(* PLC project Generated.project, CODESYS CODESYS V3.5 SP19 Patch 1 *)
(* stored: creationDateTime 2026-11-16T05:01:26.673404, modificationDateTime 2026-11-16T05:01:26.673404 *)

(* DOC: DOC/AF/AF_Partie-13_Fonction_Simulation_v2.5.md Modele dynamique M3 confine au SimBench. *)
FUNCTION_BLOCK FB_Sim_Translation
  VAR_INPUT
    Enable : BOOL;
    ReqTremie : BOOL;
    ReqMaintenance : BOOL;
    SpeedTgt_Pct : REAL;
    PosTremie_M : REAL := 0;  (* T301/L1 — SOURCE UNIQUE : le banc ne porte AUCUNE position ni echelle propre. Positions capteurs = reglages machine (GVL_PERSISTENT._TranslationPos*_M) et gain = gain EFFECTIVEMENT consomme par l'estimateur (PRG_05 FB_Translation_OdometryGain.GainActive), passes par PRG_02 -> FB_SimBench. Vitesse chariot = sens x gain x frequence. Historique : l'ancienne echelle en dur (30 m / FullTravelTimeS / 40 Hz) a diverge du gain reel (T360/T361, sauts de 4 a 9 m) — doublon supprime, gate G518 anti-retour. --> [CFG] Position capteur Tremie (m) *)
    PosPV_M : REAL := 1.5;  (* --> [CFG] Position capteur PV (m) *)
    PosP2_M : REAL := 3.5;  (* --> [CFG] Position capteur P2 (m) *)
    PosP1_M : REAL := 5;  (* --> [CFG] Position capteur P1 (m) *)
    PosMaintenance_M : REAL := 10;  (* --> [CFG] Position capteur Maintenance (m) *)
    GainMetersPerHzSec : REAL := 0.02;  (* --> [CFG] Gain odometrique effectif, m/(Hz.s) *)
    EndStopMargin_M : REAL := 0.5;  (* Distance capteur extreme -> butee mecanique (seule donnee propre au banc : physique du rail). Bornee a CST_MinEndStopMargin_M pour que le capteur extreme reste franchissable. *)
    BrakeReleaseCmd : BOOL := TRUE;
    MaxFreq_Hz : REAL := 50;  (* ECHELLE DE LA CONSIGNE. PRG_02 envoie SpeedCmd_Pct = f / 50 Hz x 100 : le simulateur reconvertit avec le MEME maximum, sinon 20 Hz reels (40 %) deviendraient 16 Hz simules. Maximum = GVL_PERSISTENT._TranslationMaxFreq_Hz (50 Hz), passe par FB_SimBench (CST_M3MaxFreq_Hz, egalite verifiee par G518). Ne pas confondre avec l'ancienne echelle (40 Hz) : echelle ODOMETRIQUE (gain 0,02 m/(Hz.s)). *)
    SpeedFactor : REAL := 1;  (* ACCELERATION DU BANC (confort d'essai). Le chariot avance SpeedFactor fois plus vite ET la frequence RETOURNEE au PLC est multipliee d'autant : l'estimateur (f x gain) suit exactement le chariot, sans saut de recalage, et le ratio publie reste 0,02 m/(Hz.s) (G518). Borne 1..5. 1,0 = dynamique reelle. Le frein et la memoire de sens restent sur la frequence physique du variateur simule. *)
    AccelRate_HzPerS : REAL := 20;
    DecelRate_HzPerS : REAL := 25;  (* pente d'arret relevee sur trace reelle (rampe variateur / rampe PLC) *)
    DriveTimeConstantS : REAL := 0.15;
    BrakeOpenDelayS : REAL := 0.1;
    BrakeCloseDelayS : REAL := 0.09;
    BrakeContactDelayS : REAL := 0.01;
    BrakeFaultCloseWhileRunning : BOOL := FALSE;  (* FAUTE EXPLICITE frein M3 — defaut FALSE : reproduit le defaut terrain « frein ferme alors que le variateur retourne encore 10,00 Hz » (trace 2026-09-04, 26,437 s, State.ErrorId=64). La garde nominale 0,5 Hz du frein n'est pas modifiee. *)
    BrakeFaultCloseDelay_S : REAL := 0;
    BrakePhysicalActive : BOOL := FALSE;  (* L3 — FREIN PHYSIQUE (2026-10-28). FALSE = historique (frein ne retombe que sous 0,5 Hz, arret instantane). TRUE = frein a manque de courant reel : retombe CloseDelay apres la coupure bobine QUELLE QUE SOIT la vitesse, puis le chariot decelere sur le frein (BrakeDecel_Mps2) ; frein serre = chariot bloque meme si le variateur pousse. defaut FB = historique ; GVL_Simulation.SimM3BrakePhysicalActive = TRUE (source unique) *)
    BrakeDecel_Mps2 : REAL := 2;  (* HYPOTHESE : 0,4 m/s (20 Hz) -> arret ~0,2 s / ~4 cm *)
    CartFreeActive : BOOL := FALSE;  (* L4 — CHARIOT LIBRE (2026-10-28). FALSE = historique (chariot esclave de la frequence). TRUE = quand le frein est OUVERT et que le variateur n'applique plus de couple (mot a 0 et rampe variateur terminee), le chariot n'est plus tenu : il garde sa vitesse et subit la poussee de la benne suspendue (rapport de masse x g x angle), la pente et le frottement de roulement. Valeurs = HYPOTHESES, sans mesure terrain. *)
    LoadMassRatio : REAL := 0.5;  (* masse benne / masse totale chariot+benne *)
    RollingFriction_Mps2 : REAL := 0.3;  (* FEM 1.001 : frottement global galets + reducteur accouple *)
    StaticFriction_Mps2 : REAL := 0.35;  (* Seuil de decollement statique (anti-pompage pendulaire) *)
    Slope_Mps2 : REAL := 0;  (* composante de pente, + vers Maintenance *)
    SensorCamDropoutActive : BOOL := FALSE;  (* L5 — came capteurs (vu -> perdu -> retrouve -> fixe), appliquee aux 5 capteurs. *)
    SensorCamDropoutStart_M : REAL := 0.02;
    SensorCamDropoutWidth_M : REAL := 0.04;
    SuspendedLoadLength_M : REAL := 1.5;
    SuspendedLoadDamping : REAL := 0.35;
    LoadReactionGain_Mps2 : REAL := 0.2;
    EndStopRecoilMax_M : REAL := 0;  (* BUTEE MECANIQUE — recul borne apres arret serre. 0.0 (defaut) conserve EXACTEMENT le comportement historique : position ET vitesse figees a la butee (decision de review tracee, correctif « contact rigide »). > 0 : l'inertie du chariot reste absorbee par la butee, MAIS la reaction de la charge peut ressortir le chariot de la zone capteur — comportement observe sur la trace terrain du 2026-09-04 a 26,437 s (Tremie actif 1 echantillon puis perdu definitivement). Valeur SYNTHETIQUE, en attente de mesure terrain. *)
    LoadFrequencyDroopGain_Hz : REAL := 0.5;
    SensorJitterAmplitude_M : REAL := 0.01;
    SensorStabilizationS : REAL := 1;
    SensorElectricalDelayS : REAL := 0.01;
    SensorIntermittenceActive : BOOL := FALSE;
    SensorLoadAngleTriggerRad : REAL := 0.01;
    SensorScenarioSeed : UDINT := 3001;
    SensorHysteresis_M : REAL := 0.02;
    SensorIntermittencePeriodS : REAL := 0.12;
    SensorBlipTransitions : UDINT := 0;  (* BLIP COURT — second profil capteur, independant du train ~1 s ci-dessus. BlipTransitions = 0 (defaut) : profil historique strictement inchange. Valeurs de trace : Tremie 1 excursion de 0,2 s (2 echantillons a 100 ms), PV 1 excursion de 0,1 s (1 echantillon). ⚠️ LIMITE CONNUE (revue 2026-09-20, F11) : UNE SEULE largeur globale est appliquee aux cinq capteurs. Les deux signatures de la trace (Tremie 0,200 s et PV 0,100 s) ne sont donc PAS rejouables dans la meme passe : il faut deux executions avec des valeurs differentes de SensorBlipDurationS. Une largeur par capteur exigerait un ARRAY[1..5] OF REAL, non retenu dans ce lot. *)
    SensorBlipDurationS : REAL := 0.2;
  END_VAR
  VAR_OUTPUT
    PosTremie : BOOL;
    PosPV : BOOL;
    PosP2 : BOOL;
    PosP1 : BOOL;
    PosMaintenance : BOOL;
    FrequencyCmd_Hz : REAL;
    ElectricalFrequency_Hz : REAL;
    ActualFrequency_Hz : REAL;
    BrakeCoilEnergized : BOOL;
    BrakeMechanicallyOpen : BOOL;
    BrakeContactOpen : BOOL;
    BrakeFaultCloseActive : BOOL;
    PositionTrue_M : REAL;
    VelocityTrue_Mps : REAL;
    LoadAngle_Rad : REAL;
    SensorPosition_M : REAL;
    SensorTransitionCount : UDINT;
    SensorBlipActive : BOOL;
    HardStopTremieActive : BOOL;
    HardStopMaintenanceActive : BOOL;
    ObsOvershootLast_M : REAL;  (* L2 — OBSERVATION (aucun effet sur le modele ni sur le programme) Distance roulee entre le 1er front du dernier capteur d'arret (Tremie, P1, Maintenance) et l'arret *)
    ObsOvershootSensorId : INT;  (* 1 = Tremie, 3 = P1, 5 = Maintenance, 0 = aucun *)
    ObsEndStopHitCount : UDINT;  (* Nombre de chocs en butee mecanique *)
    ObsEndStopImpactSpeed_Mps : REAL;  (* Vitesse au dernier choc en butee *)
    ObsBrakeClosedMovingCount : UDINT;  (* Nombre de fermetures mecaniques du frein chariot en mouvement *)
    ObsCartFree : BOOL;  (* L4 : frein ouvert ET variateur sans couple -> chariot libre *)
    ObsFreeRollLast_M : REAL;  (* L4 : distance parcourue pendant le dernier episode libre *)
  END_VAR
  VAR
    ObsArmed : BOOL;  (* Front capteur d'arret vu, arret pas encore constate *)
    ObsEdgePosition_M : REAL;  (* Position vraie au 1er front du capteur d'arret *)
    ObsPrevTremie : BOOL;
    ObsPrevP1 : BOOL;
    ObsPrevMaintenance : BOOL;
    ObsPrevBrakeOpen : BOOL;
    ObsPrevHardStop : BOOL;
    ObsSpeedBeforeStop_Mps : REAL;  (* Vitesse du scan avant le calcul de butee *)
    DriveTorqueActive : BOOL;  (* L4 : variateur commande ou encore en rampe -> chariot tenu *)
    FreeAccel_Mps2 : REAL;  (* L4 : acceleration nette du chariot libre *)
    FreeVelocity_Mps : REAL;  (* Vitesse apres integration de la force externe *)
    FrictionStep_Mps : REAL;  (* Impulsion dissipative maximale sur le pas *)
    FreeRollStart_M : REAL;  (* L4 : position au debut de l'episode libre *)
    instCycleTime : FB_CycleTime;
    Initialized : BOOL;
    DirectionSign : REAL;
    TravelDirection : REAL;  (* Sens de deplacement MEMORISE. La commande peut etre retiree AVANT l'arret physique (deceleration libre du variateur) : le sens du dernier ordre valide est conserve tant que le variateur retourne de la vitesse, puis purge a l'arret. Sans cette memoire, la vitesse du chariot s'effondrait au scan de retrait de commande alors que la frequence retournee decroit encore. ⚠️ ORDRE DE GRANDEUR NON MESURE : la trace terrain ne contient AUCUNE variable de position (15 TraceVariable : DI, frequences, mots d'etat, erreurs). La distance de roue libre de la fenetre 14,67 -> 16,16 s est donc une ESTIMATION dependante du modele d'echelle, qui vaut approximativement 1,1 a 1,3 m selon la methode d'integration retenue (gain audit 0,0551 m/(Hz.s)). A ne pas citer comme une mesure. *)
    FrequencyTarget_Hz : REAL;
    SpeedFactorApplied : REAL := 1;
    CycleTimeS : REAL;
    EndStopTremie_M : REAL;  (* butee mecanique cote Tremie = capteur Tremie - marge *)
    EndStopMaintenance_M : REAL;  (* butee mecanique cote Maintenance = capteur Maintenance + marge *)
    VelocityTarget_Mps : REAL;
    CartAcceleration_Mps2 : REAL;
    PreviousVelocity_Mps : REAL;
    PositionCandidate_M : REAL;
    RecoilMax_M : REAL;  (* Recul de butee ECRETE a la course : une valeur d'entree aberrante ne peut pas autoriser une position hors des butees (revue du 2026-09-20, F8). *)
    SensorNoiseState : REAL := 0.371;
    SensorNoise_M : REAL;
    instSensorTremie : FB_Sim_PositionSensor;
    instSensorPV : FB_Sim_PositionSensor;
    instSensorP2 : FB_Sim_PositionSensor;
    instSensorP1 : FB_Sim_PositionSensor;
    instSensorMaintenance : FB_Sim_PositionSensor;
    instDrive : FB_Sim_TranslationDrive;
    instBrake : FB_Sim_TranslationBrake;
    instSuspendedLoad : FB_Sim_SuspendedLoad;
    CST_MinEndStopMargin_M : REAL := 0.05;  (* Marge mini capteur extreme -> butee : au-dela de l'hysteresis capteur, sinon le mot 11111 / 00000 ne pourrait jamais etre produit (capteur colle a la butee). *)
    CST_StopFrequency_Hz : REAL := 0.5;  (* Meme seuil d'arret que FB_Sim_TranslationBrake.CST_StopFrequency_Hz (0,5 Hz). Valide par la trace terrain du 2026-09-04 : frein ouvert a 0,60 Hz, ferme a 0,00 Hz. *)
  END_VAR

            

instCycleTime(DefaultValueS := 0.010);
(* Le modele mono-pas suit le temps de cycle reel jusqu'a 100 ms. Cette borne
   evite de ralentir artificiellement la dynamique lorsque la trace est executee
   dans VISU_TASK (environ 100 ms), tout en restant stable pour le pendule reduit.
   Au-dela, FB_CycleTime fournit deja son temps de secours et aucun saut aberrant
   n'est accepte. La qualification des delais sub-100 ms exige toutefois une tache
   de trace plus rapide que 100 ms. *)
CycleTimeS := LIMIT(0.001, instCycleTime.CycleTimeS, 0.100);

(* Butees mecaniques derivees des capteurs extremes (reglages machine) + marge du rail. *)
EndStopTremie_M := PosTremie_M - MAX(EndStopMargin_M, CST_MinEndStopMargin_M);
EndStopMaintenance_M := PosMaintenance_M + MAX(EndStopMargin_M, CST_MinEndStopMargin_M);

IF NOT Enable THEN
    Initialized := FALSE;
    instDrive(Enable := FALSE);
    instBrake(Enable := FALSE);
    instSuspendedLoad(Enable := FALSE);
    FrequencyCmd_Hz := 0.0;
    ElectricalFrequency_Hz := 0.0;
    ActualFrequency_Hz := 0.0;
    BrakeMechanicallyOpen := FALSE;
    BrakeContactOpen := FALSE;
    BrakeCoilEnergized := FALSE;
    BrakeFaultCloseActive := FALSE;
    PositionTrue_M := PosP1_M;
    VelocityTrue_Mps := 0.0;
    PreviousVelocity_Mps := 0.0;
    TravelDirection := 0.0;
    LoadAngle_Rad := 0.0;
    SensorTransitionCount := 0;
    SensorBlipActive := FALSE;
    HardStopTremieActive := FALSE;
    HardStopMaintenanceActive := FALSE;
    (* Repli deterministe compatible avec le mot thermometre P1 = 00011. *)
    PosTremie := FALSE;
    PosPV := FALSE;
    PosP2 := FALSE;
    PosP1 := TRUE;
    PosMaintenance := TRUE;
    instSensorTremie(Enable := FALSE);
    instSensorPV(Enable := FALSE);
    instSensorP2(Enable := FALSE);
    instSensorP1(Enable := FALSE);
    instSensorMaintenance(Enable := FALSE);
    RETURN;
ELSIF NOT Initialized THEN
    Initialized := TRUE;
    PositionTrue_M := PosP1_M;
    TravelDirection := 0.0;
END_IF;

IF Enable THEN
    DirectionSign := 0.0;
    IF ReqTremie AND NOT ReqMaintenance THEN
        DirectionSign := -1.0;
    ELSIF ReqMaintenance AND NOT ReqTremie THEN
        DirectionSign := 1.0;
    END_IF;

    FrequencyTarget_Hz := LIMIT(0.0, ABS(SpeedTgt_Pct) * MaxFreq_Hz / 100.0, MaxFreq_Hz);
    IF DirectionSign = 0.0 THEN
        FrequencyTarget_Hz := 0.0;
    END_IF;
    instDrive(Enable := TRUE, FrequencyTgt_Hz := FrequencyTarget_Hz,
        AccelRate_HzPerS := AccelRate_HzPerS, DecelRate_HzPerS := DecelRate_HzPerS,
        TimeConstant_S := DriveTimeConstantS,
        LoadAngularVelocity_RadPerS := instSuspendedLoad.AngularVelocity_RadPerS,
        LoadFrequencyDroopGain_Hz := LoadFrequencyDroopGain_Hz, CycleTime_S := CycleTimeS);
    FrequencyCmd_Hz := instDrive.FrequencyCmd_Hz;
    ElectricalFrequency_Hz := instDrive.ElectricalFrequency_Hz;
    SpeedFactorApplied := LIMIT(1.0, SpeedFactor, 5.0);
    ActualFrequency_Hz := instDrive.ActualFrequency_Hz * SpeedFactorApplied;
    instBrake(Enable := TRUE, ReleaseCmd := BrakeReleaseCmd,
        ActualFrequency_Hz := instDrive.ActualFrequency_Hz, OpenDelay_S := BrakeOpenDelayS,
        CloseDelay_S := BrakeCloseDelayS, ContactDelay_S := BrakeContactDelayS,
        CycleTime_S := CycleTimeS,
        FaultCloseWhileRunning := BrakeFaultCloseWhileRunning,
        FaultCloseDelay_S := BrakeFaultCloseDelay_S,
        PhysicalBrakeActive := BrakePhysicalActive);
    BrakeCoilEnergized := instBrake.CoilEnergized;
    BrakeMechanicallyOpen := instBrake.MechanicallyOpen;
    BrakeContactOpen := instBrake.ContactOpen;
    BrakeFaultCloseActive := instBrake.FaultCloseActive;

    (* Sens memorise (C3). Regles, dans cet ordre :
       1. un ordre simple valide (re)memorise le sens ;
       2. deux ordres contradictoires neutralisent immediatement le sens — aucune
          excitation inventee (preserve TC-T300-MEC-030) ;
       3. commande retiree : le sens est CONSERVE tant que le variateur retourne de la
          vitesse (deceleration libre), puis purge des que la vitesse est nulle. *)
    IF ReqTremie AND NOT ReqMaintenance THEN
        TravelDirection := -1.0;
    ELSIF ReqMaintenance AND NOT ReqTremie THEN
        TravelDirection := 1.0;
    ELSIF ReqTremie AND ReqMaintenance THEN
        TravelDirection := 0.0;
    ELSIF ABS(instDrive.ActualFrequency_Hz) <= CST_StopFrequency_Hz THEN
        TravelDirection := 0.0;
    END_IF;

    PreviousVelocity_Mps := VelocityTrue_Mps;
    IF BrakeMechanicallyOpen THEN
        (* Source unique : meme gain que l'estimateur machine (vitesse = gain x frequence). *)
        VelocityTarget_Mps := TravelDirection * MAX(0.0, GainMetersPerHzSec) * ActualFrequency_Hz;
    ELSE
        VelocityTarget_Mps := 0.0;
    END_IF;
    (* L4 : le variateur tient le chariot tant qu'il est commande ou que sa SORTIE electrique
       alimente encore le moteur (rampe + reponse) ; ensuite, plus aucun couple.
       Reprise de commande en roue libre : pas de reprise a la volee (le variateur repart de 0 Hz). *)
    DriveTorqueActive := (DirectionSign <> 0.0) OR (instDrive.ElectricalFrequency_Hz > CST_StopFrequency_Hz);
    ObsCartFree := CartFreeActive AND BrakeMechanicallyOpen AND NOT DriveTorqueActive;
    IF ObsCartFree THEN
        (* Poussee de la benne (angle du scan precedent) + pente - frottement oppose au mouvement. *)
        (* Pendule sur chariot libre : x'' = m_benne / m_chariot x g x theta = r / (1 - r) x g x theta. *)
        FreeAccel_Mps2 := (LIMIT(0.0, LoadMassRatio, 0.9) / (1.0 - LIMIT(0.0, LoadMassRatio, 0.9)))
                          * 9.81 * instSuspendedLoad.Angle_Rad + Slope_Mps2;
        IF ABS(VelocityTrue_Mps) < 0.001 THEN
            (* Adherence statique au repos : ne decolle que si la poussee depasse le frottement statique *)
            IF ABS(FreeAccel_Mps2) <= MAX(0.0, StaticFriction_Mps2) THEN
                FreeAccel_Mps2 := 0.0;
                VelocityTrue_Mps := 0.0;
            ELSIF FreeAccel_Mps2 > 0.0 THEN
                FreeAccel_Mps2 := FreeAccel_Mps2 - MAX(0.0, StaticFriction_Mps2);
            ELSE
                FreeAccel_Mps2 := FreeAccel_Mps2 + MAX(0.0, StaticFriction_Mps2);
            END_IF;
            VelocityTrue_Mps := VelocityTrue_Mps + FreeAccel_Mps2 * CycleTimeS;
        ELSE
            (* La force externe peut inverser le mouvement ; le frottement ne peut
               que reduire sa vitesse, au plus jusqu'a zero. *)
            FreeVelocity_Mps := VelocityTrue_Mps + FreeAccel_Mps2 * CycleTimeS;
            FrictionStep_Mps := MAX(0.0, RollingFriction_Mps2) * CycleTimeS;
            IF (((VelocityTrue_Mps > 0.0) AND (FreeVelocity_Mps <= 0.0))
                OR ((VelocityTrue_Mps < 0.0) AND (FreeVelocity_Mps >= 0.0)))
                AND (ABS(FreeAccel_Mps2) <= MAX(0.0, StaticFriction_Mps2)) THEN
                (* Passage par zero pendant le pas : l'adherence interdit un redemarrage
                   sous le seuil statique, meme si la force est opposee au mouvement. *)
                VelocityTrue_Mps := 0.0;
            ELSIF FreeVelocity_Mps > 0.0 THEN
                VelocityTrue_Mps := MAX(0.0, FreeVelocity_Mps - FrictionStep_Mps);
            ELSE
                VelocityTrue_Mps := MIN(0.0, FreeVelocity_Mps + FrictionStep_Mps);
            END_IF;
        END_IF;
    ELSIF BrakeMechanicallyOpen THEN
        (* Vitesse suivant directement le variateur (deja filtre par instDrive) sans double PT1 *)
        VelocityTrue_Mps := VelocityTarget_Mps;
    ELSIF BrakePhysicalActive THEN
        (* L3 : frein serre -> deceleration sur le frein jusqu'a l'arret, puis chariot bloque. *)
        IF VelocityTrue_Mps > 0.0 THEN
            VelocityTrue_Mps := MAX(0.0, VelocityTrue_Mps - MAX(0.0, BrakeDecel_Mps2) * CycleTimeS);
        ELSE
            VelocityTrue_Mps := MIN(0.0, VelocityTrue_Mps + MAX(0.0, BrakeDecel_Mps2) * CycleTimeS);
        END_IF;
    ELSE
        VelocityTrue_Mps := 0.0;   (* historique : arret instantane *)
    END_IF;
    ObsSpeedBeforeStop_Mps := VelocityTrue_Mps;
    HardStopTremieActive := FALSE;
    HardStopMaintenanceActive := FALSE;
    PositionCandidate_M := PositionTrue_M + VelocityTrue_Mps * CycleTimeS;
    IF PositionCandidate_M < EndStopTremie_M THEN
        PositionTrue_M := EndStopTremie_M;
        VelocityTrue_Mps := 0.0;
        HardStopTremieActive := TRUE;
    ELSIF PositionCandidate_M > EndStopMaintenance_M THEN
        PositionTrue_M := EndStopMaintenance_M;
        VelocityTrue_Mps := 0.0;
        HardStopMaintenanceActive := TRUE;
    END_IF;
    CartAcceleration_Mps2 := (VelocityTrue_Mps - PreviousVelocity_Mps) / CycleTimeS;
    instSuspendedLoad(Enable := TRUE, BrakeMechanicallyOpen := BrakeMechanicallyOpen,
        CartAcceleration_Mps2 := CartAcceleration_Mps2, Length_M := SuspendedLoadLength_M,
        Damping := SuspendedLoadDamping, ReactionGain_Mps2 := LoadReactionGain_Mps2,
        CycleTime_S := CycleTimeS);
    LoadAngle_Rad := instSuspendedLoad.Angle_Rad;
    IF HardStopTremieActive OR HardStopMaintenanceActive THEN
        RecoilMax_M := MIN(MAX(0.0, EndStopRecoilMax_M), EndStopMaintenance_M - EndStopTremie_M);
        IF (RecoilMax_M > 0.0) AND BrakeMechanicallyOpen THEN
            (* Recul autorise UNIQUEMENT en s'eloignant de la butee touchee, borne par
               EndStopRecoilMax_M : jamais plus loin dans la butee, jamais de saut cache. *)
            VelocityTrue_Mps := VelocityTrue_Mps + instSuspendedLoad.VelocityReaction_Mps;
            (* Contre une butee, l'entrainement DECROCHE : il ne maintient pas une consigne de
               vitesse dans l'obstacle. Sans cette purge, la consigne de vitesse ecrasait en
               permanence la reaction de charge et le chariot ne pouvait jamais ressortir de
               la zone capteur (recul alors impossible, quelle que soit la charge). *)
            TravelDirection := 0.0;
            IF HardStopTremieActive THEN
                VelocityTrue_Mps := MAX(0.0, VelocityTrue_Mps);
                PositionCandidate_M := LIMIT(EndStopTremie_M,
                    PositionTrue_M + VelocityTrue_Mps * CycleTimeS,
                    EndStopTremie_M + RecoilMax_M);
            ELSE
                VelocityTrue_Mps := MIN(0.0, VelocityTrue_Mps);
                PositionCandidate_M := LIMIT(EndStopMaintenance_M - RecoilMax_M,
                    PositionTrue_M + VelocityTrue_Mps * CycleTimeS,
                    EndStopMaintenance_M);
            END_IF;
            PositionTrue_M := PositionCandidate_M;
        ELSE
            VelocityTrue_Mps := 0.0;
        END_IF;
    ELSE
        IF NOT ObsCartFree THEN
            (* Reaction historique (negligeable) ; en mode libre la poussee est deja integree (L4). *)
            VelocityTrue_Mps := VelocityTrue_Mps + instSuspendedLoad.VelocityReaction_Mps;
        END_IF;
        PositionCandidate_M := PositionTrue_M + VelocityTrue_Mps * CycleTimeS;
        IF PositionCandidate_M < EndStopTremie_M THEN
            PositionTrue_M := EndStopTremie_M;
            VelocityTrue_Mps := 0.0;
            HardStopTremieActive := TRUE;
        ELSIF PositionCandidate_M > EndStopMaintenance_M THEN
            PositionTrue_M := EndStopMaintenance_M;
            VelocityTrue_Mps := 0.0;
            HardStopMaintenanceActive := TRUE;
        ELSE
            PositionTrue_M := PositionCandidate_M;
        END_IF;
    END_IF;
END_IF;

IF Enable AND (ABS(LoadAngle_Rad) > 0.0001) THEN
    SensorNoiseState := 3.91 * SensorNoiseState * (1.0 - SensorNoiseState);
    SensorNoise_M := (2.0 * SensorNoiseState - 1.0) * SensorJitterAmplitude_M;
ELSE
    SensorNoise_M := 0.0;
END_IF;
(* Les capteurs sont fixes au rail et observent le chariot. Le balancier agit
   seulement par la reaction mecanique sur PositionTrue_M et conditionne un
   episode electrique ; aucune deflexion de godet n'est injectee directement. *)
SensorPosition_M := PositionTrue_M + SensorNoise_M;
(* Les capteurs M3 sont volontairement cumulatifs : 11111 -> 00000. Chaque
   brique garde son hysteresis et son episode propres ; aucun timer partage ne
   peut masquer un front d'un autre capteur. *)
instSensorTremie(Enable := Enable, Position_M := SensorPosition_M,
    Threshold_M := PosTremie_M, Hysteresis_M := SensorHysteresis_M,
    ElectricalDelayS := SensorElectricalDelayS, IntermittenceActive := SensorIntermittenceActive
        AND (ABS(LoadAngle_Rad) >= SensorLoadAngleTriggerRad),
    IntermittenceDurationS := SensorStabilizationS, IntermittencePeriodS := SensorIntermittencePeriodS,
    ScenarioSeed := SensorScenarioSeed + 11,
    BlipTransitions := SensorBlipTransitions, BlipDurationS := SensorBlipDurationS,
    CamDropoutActive := SensorCamDropoutActive, CamDropoutStart_M := SensorCamDropoutStart_M,
    CamDropoutWidth_M := SensorCamDropoutWidth_M,
    FiniteCamActive := TRUE, CamLength_M := 0.04,
    CycleTimeS := CycleTimeS);
instSensorPV(Enable := Enable, Position_M := SensorPosition_M,
    Threshold_M := PosPV_M, Hysteresis_M := SensorHysteresis_M,
    ElectricalDelayS := SensorElectricalDelayS, IntermittenceActive := SensorIntermittenceActive
        AND (ABS(LoadAngle_Rad) >= SensorLoadAngleTriggerRad),
    IntermittenceDurationS := SensorStabilizationS, IntermittencePeriodS := SensorIntermittencePeriodS,
    ScenarioSeed := SensorScenarioSeed + 23,
    BlipTransitions := SensorBlipTransitions, BlipDurationS := SensorBlipDurationS,
    CamDropoutActive := SensorCamDropoutActive, CamDropoutStart_M := SensorCamDropoutStart_M,
    CamDropoutWidth_M := SensorCamDropoutWidth_M,
    CycleTimeS := CycleTimeS);
instSensorP2(Enable := Enable, Position_M := SensorPosition_M,
    Threshold_M := PosP2_M, Hysteresis_M := SensorHysteresis_M,
    ElectricalDelayS := SensorElectricalDelayS, IntermittenceActive := SensorIntermittenceActive
        AND (ABS(LoadAngle_Rad) >= SensorLoadAngleTriggerRad),
    IntermittenceDurationS := SensorStabilizationS, IntermittencePeriodS := SensorIntermittencePeriodS,
    ScenarioSeed := SensorScenarioSeed + 37,
    BlipTransitions := SensorBlipTransitions, BlipDurationS := SensorBlipDurationS,
    CamDropoutActive := SensorCamDropoutActive, CamDropoutStart_M := SensorCamDropoutStart_M,
    CamDropoutWidth_M := SensorCamDropoutWidth_M,
    CycleTimeS := CycleTimeS);
instSensorP1(Enable := Enable, Position_M := SensorPosition_M,
    Threshold_M := PosP1_M, Hysteresis_M := SensorHysteresis_M,
    ElectricalDelayS := SensorElectricalDelayS, IntermittenceActive := SensorIntermittenceActive
        AND (ABS(LoadAngle_Rad) >= SensorLoadAngleTriggerRad),
    IntermittenceDurationS := SensorStabilizationS, IntermittencePeriodS := SensorIntermittencePeriodS,
    ScenarioSeed := SensorScenarioSeed + 53,
    BlipTransitions := SensorBlipTransitions, BlipDurationS := SensorBlipDurationS,
    CamDropoutActive := SensorCamDropoutActive, CamDropoutStart_M := SensorCamDropoutStart_M,
    CamDropoutWidth_M := SensorCamDropoutWidth_M,
    CycleTimeS := CycleTimeS);
instSensorMaintenance(Enable := Enable, Position_M := SensorPosition_M,
    Threshold_M := PosMaintenance_M, Hysteresis_M := SensorHysteresis_M,
    ElectricalDelayS := SensorElectricalDelayS, IntermittenceActive := SensorIntermittenceActive
        AND (ABS(LoadAngle_Rad) >= SensorLoadAngleTriggerRad),
    IntermittenceDurationS := SensorStabilizationS, IntermittencePeriodS := SensorIntermittencePeriodS,
    ScenarioSeed := SensorScenarioSeed + 71,
    BlipTransitions := SensorBlipTransitions, BlipDurationS := SensorBlipDurationS,
    CamDropoutActive := SensorCamDropoutActive, CamDropoutStart_M := SensorCamDropoutStart_M,
    CamDropoutWidth_M := SensorCamDropoutWidth_M,
    CycleTimeS := CycleTimeS);

PosTremie := instSensorTremie.ElectricalOutput;
PosPV := instSensorPV.ElectricalOutput;
PosP2 := instSensorP2.ElectricalOutput;
PosP1 := instSensorP1.ElectricalOutput;
PosMaintenance := instSensorMaintenance.ElectricalOutput;
SensorTransitionCount := instSensorTremie.TransitionCount + instSensorPV.TransitionCount
    + instSensorP2.TransitionCount + instSensorP1.TransitionCount
    + instSensorMaintenance.TransitionCount;
SensorBlipActive := instSensorTremie.BlipActive OR instSensorPV.BlipActive
    OR instSensorP2.BlipActive OR instSensorP1.BlipActive
    OR instSensorMaintenance.BlipActive;

(* ── L2 OBSERVATION (lecture seule, aucun effet sur le modele) ───────────────────────── *)
IF Enable THEN
    (* Frein serre en mouvement : front de fermeture mecanique avec vitesse non nulle. *)
    IF ObsPrevBrakeOpen AND NOT BrakeMechanicallyOpen AND (ABS(PreviousVelocity_Mps) > 0.03) THEN
        ObsBrakeClosedMovingCount := ObsBrakeClosedMovingCount + 1;
    END_IF;
    ObsPrevBrakeOpen := BrakeMechanicallyOpen;

    (* Choc en butee : front de HardStop, vitesse avant contact. *)
    IF (HardStopTremieActive OR HardStopMaintenanceActive) AND NOT ObsPrevHardStop THEN
        ObsEndStopHitCount := ObsEndStopHitCount + 1;
        ObsEndStopImpactSpeed_Mps := ABS(ObsSpeedBeforeStop_Mps);
    END_IF;
    ObsPrevHardStop := HardStopTremieActive OR HardStopMaintenanceActive;

    (* Depassement : 1er front d'un capteur d'arret (Tremie montant, P1 dans les deux sens,
       Maintenance descendant) -> position memorisee ; les rebonds du MEME capteur sont ignores
       tant que l'arret n'est pas constate ; un autre capteur franchi remplace le repere. *)
    (* Armement seulement chariot en mouvement : un rebond capteur a l'arret n'ecrase pas la mesure. *)
    IF ABS(VelocityTrue_Mps) <= 0.005 THEN
        ObsArmed := ObsArmed;   (* chariot a l'arret : aucun armement *)
    ELSIF (PosTremie AND NOT ObsPrevTremie) AND NOT (ObsArmed AND ObsOvershootSensorId = 1) THEN
        ObsArmed := TRUE; ObsOvershootSensorId := 1; ObsEdgePosition_M := PositionTrue_M;
    ELSIF (PosP1 <> ObsPrevP1) AND NOT (ObsArmed AND ObsOvershootSensorId = 3) THEN
        ObsArmed := TRUE; ObsOvershootSensorId := 3; ObsEdgePosition_M := PositionTrue_M;
    ELSIF (ObsPrevMaintenance AND NOT PosMaintenance) AND NOT (ObsArmed AND ObsOvershootSensorId = 5) THEN
        ObsArmed := TRUE; ObsOvershootSensorId := 5; ObsEdgePosition_M := PositionTrue_M;
    END_IF;
    ObsPrevTremie := PosTremie;
    ObsPrevP1 := PosP1;
    ObsPrevMaintenance := PosMaintenance;

    (* L4 : distance de l'episode libre (frein ouvert, variateur sans couple). *)
    IF NOT ObsCartFree THEN
        FreeRollStart_M := PositionTrue_M;
    ELSE
        ObsFreeRollLast_M := ABS(PositionTrue_M - FreeRollStart_M);
    END_IF;

    IF ObsArmed AND (ABS(VelocityTrue_Mps) < 0.001) THEN
        ObsOvershootLast_M := ABS(PositionTrue_M - ObsEdgePosition_M);
        ObsArmed := FALSE;
    END_IF;
END_IF;

          
END_FUNCTION_BLOCK

(* ======================================================================= ⚙️ FB_CycleTime — Mesure du temps de cycle réel de la tâche ─────────────────────────────────────────────────────────────── 🎯 Rôle : Calcul du dt réel entre deux exécutions successives ⚙️ Calcul : Delta horloge système TIME() converti en secondes 🛡️ Robustesse : dt borné (0 < dt <= CST_MaxCycleDeltaMs) sinon valeur de secours — neutralise les artefacts de rebouclage TIME() (49,7 j) et de reprise (online-change, debug) 📄 Doc métier : DOC/AF/AF_Partie-03_Contrats_Composants/FB_CycleTime_v1.0.md ======================================================================= *)
FUNCTION_BLOCK FB_CycleTime
  VAR_INPUT
    DefaultValueS : REAL := 0.004;  (* === REGLAGES DE SECOURS === --> [CFG] Valeur de secours par defaut (ex: 4ms = 0.004s) *)
  END_VAR
  VAR_OUTPUT
    CycleTimeS : REAL;  (* === MESURE ET DIAGNOSTIC === <-- [DIAG] Temps ecoule reel calcule (secondes) *)
  END_VAR
  VAR
    TimeCurrent : TIME;  (* === HORLOGE ET MEMOIRE TEMPORELLE === . [LOC] Temps systeme actuel *)
    TimeLast : TIME;  (* . [LOC] Empreinte de temps du cycle precedent *)
    DeltaTimeMs : UDINT;  (* . [LOC] Ecart brut calcule (ms) *)
    InitDone : BOOL;  (* . [LOC] Drapeau d'initialisation du premier cycle *)
    CST_MaxCycleDeltaMs : UDINT := 1000;  (* === BORNE HAUTE DU DELTA DE CYCLE === Plafond physique du dt entre deux scans (ms) : au-dela -> valeur de secours *)
  END_VAR

            

{region "§1 Acquisition temps"}
// 1. ACQUISITION DU TEMPS SYSTÈME
TimeCurrent := TIME();
{endregion}

{region "§2 Initialisation"}
// 2. INITIALISATION UNIQUE AU PREMIER CYCLE
IF NOT InitDone THEN
    TimeLast := TimeCurrent;
    InitDone := TRUE;
    CycleTimeS := DefaultValueS;
    RETURN;
END_IF;
{endregion}

{region "§3 Calcul delta"}
// 3. CALCUL DU DELTA EN MILLISECONDES
DeltaTimeMs := TIME_TO_UDINT(TimeCurrent - TimeLast);
{endregion}

{region "§4 Conversion, secours et bornage"}
// 4. CONVERSION EN SECONDES, AVEC DOUBLE BORNAGE DU DELTA
//
// TIME() est un compteur systeme 32 bits en millisecondes depuis le demarrage de
// l'automate. Il n'est PAS absolu : il reboucle a 0 tous les 2^32 ms (~49,7 jours).
// La soustraction TimeCurrent - TimeLast est modulo 2^32 : au passage du rebouclage,
// tant que l'ecart reel entre deux scans reste < 49,7 j (toujours vrai a 10 ms),
// DeltaTimeMs reste correct. Le rebouclage seul n'est donc pas le risque principal.
//
// Le vrai risque est un DeltaTimeMs REELLEMENT > CST_MaxCycleDeltaMs : reprise apres
// un online-change, sortie d'un point d'arret / pas-a-pas debug, ou fenetre du
// rebouclage TIME(). Le chien de garde tache (200 ms, sensibilite 1) borne deja les
// gels en fonctionnement ; ce plafond couvre les cas hors surveillance.
// Un dt aberrant publie tel quel donnerait un CycleTimeS enorme, propage en un seul
// scan dans les rampes de vitesse et les integrateurs de position/frein -> saut
// physique. Fail-safe : hors de la plage nominale (0 < dt <= plafond), on publie la
// valeur de secours DefaultValueS au lieu de l'artefact. Pas de redemarrage auto.
//
// Borne basse dt = 0 (anti-zero, ex. premier appel du scan) et borne haute
// dt > CST_MaxCycleDeltaMs (anti-artefact) partagent la meme branche de secours.
IF (DeltaTimeMs > 0) AND (DeltaTimeMs <= CST_MaxCycleDeltaMs) THEN
    CycleTimeS := UDINT_TO_REAL(DeltaTimeMs) / 1000.0;
ELSE
    CycleTimeS := DefaultValueS;
END_IF;
{endregion}

{region "§5 Archivage"}
// 5. ARCHIVAGE POUR LE PROCHAIN CYCLE
TimeLast := TimeCurrent;
{endregion}

          
END_FUNCTION_BLOCK

(* DOC: DOC/AF/AF_Partie-13_Fonction_Simulation_v2.5.md Capteur de position cumulatif avec hysteresis et episode intermittent rejouable. Cette brique ne connait ni le mouvement ni la logique M3 : elle transforme uniquement une position mecanique vraie en DI. *)
FUNCTION_BLOCK FB_Sim_PositionSensor
  VAR_INPUT
    Enable : BOOL;
    Position_M : REAL;
    Threshold_M : REAL;
    Hysteresis_M : REAL := 0.02;
    ActiveBelowThreshold : BOOL := TRUE;
    ElectricalDelayS : REAL := 0;
    IntermittenceActive : BOOL := FALSE;
    IntermittenceDurationS : REAL := 1;
    IntermittencePeriodS : REAL := 0.12;
    ScenarioSeed : UDINT := 1;
    CycleTimeS : REAL := 0.01;
    BlipTransitions : UDINT := 0;  (* Profil « BLIP COURT » — SECOND profil, independant du train de bascules du profil d'intermittence ci-dessus (dont les parametres restent inchanges). 0 = desactive : le comportement historique est strictement conserve. Rejoue les excursions electriques courtes mesurees sur la trace terrain du 2026-09-04 : Tremie contradictoire pendant 2 echantillons a 12,24 s (~200 ms) et PV reactive 1 echantillon a 14,94 s (~100 ms). BlipTransitions = nombre de bascules electriques (1 = une excursion puis retour) ; BlipDurationS = duree de maintien de chaque etat, donc largeur de l'excursion. *)
    BlipDurationS : REAL := 0.2;
    CamDropoutActive : BOOL := FALSE;  (* L5 (2026-10-28) — MECANISME DE CAME, SPATIAL : en franchissant le capteur on le VOIT, on le PERD sur une courte zone, on le RETROUVE, puis il reste FIXE. Lie a la POSITION (pas au temps) : se produit a chaque passage, dans les DEUX sens, et reste stable a l'arret (bornes de la zone avec hysteresis CST_CamHysteresis_M contre le bruit/balancement). Zone de perte placee APRES le front de detection (cote -/+ Hysteresis_M) : [front - Start - Width ; front - Start] cote detection. FALSE = historique strictement inchange. Valeurs = HYPOTHESES. *)
    CamDropoutStart_M : REAL := 0.02;
    CamDropoutWidth_M : REAL := 0.04;
    FiniteCamActive : BOOL := FALSE;  (* Came finie : FALSE = capteur cumulatif ; TRUE = sortie active uniquement sur CamLength_M apres Threshold_M. *)
    CamLength_M : REAL := 0;
  END_VAR
  VAR_OUTPUT
    RawDetected : BOOL;
    ElectricalOutput : BOOL;
    EpisodeActive : BOOL;
    BlipActive : BOOL;
    TransitionCount : UDINT;
    EpisodeTogglePeriodS : REAL;
  END_VAR
  VAR
    Initialized : BOOL;
    PreviousRawDetected : BOOL;
    EpisodeTarget : BOOL;
    DelayTimerS : REAL;
    EpisodeTimerS : REAL;
    ToggleTimerS : REAL;
    RandomState : UDINT;
    BlipRunning : BOOL;
    BlipTimerS : REAL;
    BlipCount : UDINT;
    HystDetected : BOOL;  (* L5 : etat mecanique avec hysteresis (avant perte de came) *)
    InCamDropout : BOOL;  (* L5 : position dans la zone de perte de la came *)
    CamNear_M : REAL;  (* L5 : borne de la zone cote front de detection *)
    CamFar_M : REAL;  (* L5 : borne de la zone cote interieur *)
    PastFiniteCam : BOOL;  (* Depassement au-dela de la longueur physique de came *)
    CamEnd_M : REAL;  (* Borne de fin de came finie *)
    CST_BlipMaxTransitions : UDINT := 1000;  (* Plafond du nombre de bascules du profil « blip court » : borne la duree de l'episode et interdit tout rebouclage de compteur UDINT (revue du 2026-09-20, F9). *)
    CST_CamHysteresis_M : REAL := 0.01;  (* L5 : hysteresis des bornes de la zone de perte *)
  END_VAR

            

IF NOT Enable THEN
    Initialized := FALSE;
    RawDetected := FALSE;
    ElectricalOutput := FALSE;
    PreviousRawDetected := FALSE;
    EpisodeActive := FALSE;
    BlipActive := FALSE;
    BlipRunning := FALSE;
    BlipTimerS := 0.0;
    BlipCount := 0;
    DelayTimerS := 0.0;
    EpisodeTimerS := 0.0;
    ToggleTimerS := 0.0;
    TransitionCount := 0;
    EpisodeTogglePeriodS := 0.0;
    PastFiniteCam := FALSE;
    RETURN;
END_IF;

(* Hysteresis sur une frontiere cumulative : les cinq DI restent compatibles avec
   le mot thermometre du decodeur M3, contrairement a cinq fenetres independantes. *)
IF NOT Initialized THEN
    IF ActiveBelowThreshold THEN
        RawDetected := Position_M <= Threshold_M;
        IF FiniteCamActive THEN
            PastFiniteCam := Position_M < (Threshold_M - MAX(0.0, CamLength_M));
            RawDetected := RawDetected AND NOT PastFiniteCam;
        ELSE
            PastFiniteCam := FALSE;
        END_IF;
    ELSE
        RawDetected := Position_M >= Threshold_M;
        IF FiniteCamActive THEN
            PastFiniteCam := Position_M > (Threshold_M + MAX(0.0, CamLength_M));
            RawDetected := RawDetected AND NOT PastFiniteCam;
        ELSE
            PastFiniteCam := FALSE;
        END_IF;
    END_IF;
    HystDetected := RawDetected;
    ElectricalOutput := RawDetected;
    PreviousRawDetected := RawDetected;
    RandomState := ScenarioSeed MOD 1000000;
    IF RandomState = 0 THEN
        RandomState := 1;
    END_IF;
    EpisodeTogglePeriodS := MAX(0.01, IntermittencePeriodS);
    Initialized := TRUE;
    RETURN;
END_IF;

IF ActiveBelowThreshold THEN
    IF HystDetected THEN
        HystDetected := Position_M <= (Threshold_M + MAX(0.0, Hysteresis_M));
    ELSE
        HystDetected := Position_M <= (Threshold_M - MAX(0.0, Hysteresis_M));
    END_IF;
    (* Zone de perte : apres le front d'entree en detection (cote - hysteresis), vers l'interieur. *)
    CamNear_M := Threshold_M - MAX(0.0, Hysteresis_M) - MAX(0.0, CamDropoutStart_M);
    CamFar_M := CamNear_M - MAX(0.0, CamDropoutWidth_M);
    IF NOT CamDropoutActive THEN
        InCamDropout := FALSE;
    ELSIF InCamDropout THEN
        InCamDropout := (Position_M <= CamNear_M + CST_CamHysteresis_M) AND (Position_M > CamFar_M - CST_CamHysteresis_M);
    ELSE
        InCamDropout := (Position_M <= CamNear_M - CST_CamHysteresis_M) AND (Position_M > CamFar_M + CST_CamHysteresis_M);
    END_IF;
    CamEnd_M := Threshold_M - MAX(0.0, CamLength_M);
    IF NOT FiniteCamActive THEN
        PastFiniteCam := FALSE;
    ELSIF PastFiniteCam THEN
        PastFiniteCam := Position_M < (CamEnd_M + CST_CamHysteresis_M);
    ELSE
        PastFiniteCam := Position_M < CamEnd_M;
    END_IF;
ELSE
    IF HystDetected THEN
        HystDetected := Position_M >= (Threshold_M - MAX(0.0, Hysteresis_M));
    ELSE
        HystDetected := Position_M >= (Threshold_M + MAX(0.0, Hysteresis_M));
    END_IF;
    CamNear_M := Threshold_M + MAX(0.0, Hysteresis_M) + MAX(0.0, CamDropoutStart_M);
    CamFar_M := CamNear_M + MAX(0.0, CamDropoutWidth_M);
    IF NOT CamDropoutActive THEN
        InCamDropout := FALSE;
    ELSIF InCamDropout THEN
        InCamDropout := (Position_M >= CamNear_M - CST_CamHysteresis_M) AND (Position_M < CamFar_M + CST_CamHysteresis_M);
    ELSE
        InCamDropout := (Position_M >= CamNear_M + CST_CamHysteresis_M) AND (Position_M < CamFar_M - CST_CamHysteresis_M);
    END_IF;
    CamEnd_M := Threshold_M + MAX(0.0, CamLength_M);
    IF NOT FiniteCamActive THEN
        PastFiniteCam := FALSE;
    ELSIF PastFiniteCam THEN
        PastFiniteCam := Position_M > (CamEnd_M - CST_CamHysteresis_M);
    ELSE
        PastFiniteCam := Position_M > CamEnd_M;
    END_IF;
END_IF;
(* L5 : perte de came + came finie ; hors options, RawDetected = HystDetected. *)
RawDetected := HystDetected AND NOT InCamDropout AND NOT PastFiniteCam;

(* Un episode est declenche par un franchissement mecanique, pas par une de ses
   propres bascules electriques. Les fronts restent donc bornes et reproductibles. *)
IF RawDetected <> PreviousRawDetected THEN
    PreviousRawDetected := RawDetected;
    EpisodeTarget := RawDetected;
    (* Une bascule mecanique pendant l'episode modifie seulement la cible finale.
       Elle ne remet jamais son chronometre a zero : l'episode reste borne. *)
    IF NOT EpisodeActive THEN
        DelayTimerS := 0.0;
        EpisodeTimerS := 0.0;
        ToggleTimerS := 0.0;
        (* Tirage unique par episode : reproductible pour une graine et sans bruit
           blanc scan-par-scan. La periode varie de 70 % a 130 % du nominal. *)
        RandomState := RandomState + 7919;
        IF RandomState >= 1000000 THEN
            RandomState := RandomState - 1000000;
        END_IF;
        EpisodeTogglePeriodS := MAX(0.01, IntermittencePeriodS
            * (0.7 + UDINT_TO_REAL(RandomState MOD 6000) / 10000.0));
        EpisodeActive := IntermittenceActive AND (IntermittenceDurationS > 0.0);
    END_IF;
    (* Blip court : arme sur le meme front MECANIQUE. Ses propres bascules electriques ne
       peuvent donc jamais le rearmer — meme protection que l'episode d'intermittence. *)
    IF (BlipTransitions > 0) AND (BlipDurationS > 0.0) THEN
        BlipRunning := TRUE;
        BlipTimerS := 0.0;
        BlipCount := 0;
        BlipActive := TRUE;
        (* Ecretage : au-dela de ce plafond, un compteur UDINT pourrait reboucler et rendre
           le blip non terminant (revue du 2026-09-20, F9). *)
        BlipTransitions := MIN(BlipTransitions, CST_BlipMaxTransitions);
    END_IF;
END_IF;

IF BlipRunning THEN
    (* Protocole du blip court : (0) la sortie rejoint d'abord l'etat MECANIQUE — le
       comportement nominal reste donc visible ; puis une excursion contradictoire toutes
       les BlipDurationS, donc de largeur BlipDurationS ; enfin la sortie est rendue a
       l'etat mecanique. Nombre d'excursions = BlipTransitions. *)
    BlipTimerS := BlipTimerS + CycleTimeS;
    IF BlipTimerS >= MAX(CycleTimeS, BlipDurationS) THEN
        BlipTimerS := 0.0;
        IF BlipCount = 0 THEN
            IF ElectricalOutput <> RawDetected THEN
                ElectricalOutput := RawDetected;
                TransitionCount := TransitionCount + 1;
            END_IF;
            BlipCount := 1;
        ELSIF BlipCount <= BlipTransitions THEN
            ElectricalOutput := NOT ElectricalOutput;
            TransitionCount := TransitionCount + 1;
            BlipCount := BlipCount + 1;
        ELSE
            BlipRunning := FALSE;
            BlipActive := FALSE;
            IF ElectricalOutput <> RawDetected THEN
                ElectricalOutput := RawDetected;
                TransitionCount := TransitionCount + 1;
            END_IF;
            DelayTimerS := 0.0;
        END_IF;
    END_IF;
ELSIF EpisodeActive THEN
    EpisodeTimerS := EpisodeTimerS + CycleTimeS;
    ToggleTimerS := ToggleTimerS + CycleTimeS;
    IF ToggleTimerS >= EpisodeTogglePeriodS THEN
        ElectricalOutput := NOT ElectricalOutput;
        ToggleTimerS := 0.0;
        TransitionCount := TransitionCount + 1;
    END_IF;
    IF EpisodeTimerS >= IntermittenceDurationS THEN
        EpisodeActive := FALSE;
        IF ElectricalOutput <> EpisodeTarget THEN
            ElectricalOutput := EpisodeTarget;
            TransitionCount := TransitionCount + 1;
        END_IF;
        DelayTimerS := 0.0;
    END_IF;
ELSIF ElectricalOutput <> RawDetected THEN
    DelayTimerS := DelayTimerS + CycleTimeS;
    IF DelayTimerS >= MAX(0.0, ElectricalDelayS) THEN
        ElectricalOutput := RawDetected;
        DelayTimerS := 0.0;
        TransitionCount := TransitionCount + 1;
    END_IF;
ELSE
    DelayTimerS := 0.0;
END_IF;

          
END_FUNCTION_BLOCK

(* DOC: DOC/AF/AF_Partie-13_Fonction_Simulation_v2.5.md Pendule reduit : reaction sur chariot sans injection DI directe. *)
FUNCTION_BLOCK FB_Sim_SuspendedLoad
  VAR_INPUT
    Enable : BOOL;
    BrakeMechanicallyOpen : BOOL;
    CartAcceleration_Mps2 : REAL;
    Length_M : REAL := 1.5;
    Damping : REAL := 0.35;
    ReactionGain_Mps2 : REAL := 0.2;
    CycleTime_S : REAL := 0.01;
  END_VAR
  VAR_OUTPUT
    Ready : BOOL;
    Angle_Rad : REAL;
    AngularVelocity_RadPerS : REAL;
    VelocityReaction_Mps : REAL;
  END_VAR
  VAR
    AngularAccel_RadPerS2 : REAL;
    CST_Gravity_Mps2 : REAL := 9.81;
    CST_MinLength_M : REAL := 0.1;
    CST_MaxAngle_Rad : REAL := 0.6;
    CST_MaxAngularVelocity_RadPerS : REAL := 4;
  END_VAR

            

IF NOT Enable THEN
    Ready := FALSE;
    Angle_Rad := 0.0;
    AngularVelocity_RadPerS := 0.0;
    VelocityReaction_Mps := 0.0;
    RETURN;
END_IF;

VelocityReaction_Mps := 0.0;
IF Length_M > CST_MinLength_M THEN
    AngularAccel_RadPerS2 := -(CST_Gravity_Mps2 / Length_M) * Angle_Rad
        - MAX(0.0, Damping) * AngularVelocity_RadPerS
        - CartAcceleration_Mps2 / Length_M;
    AngularVelocity_RadPerS := LIMIT(-CST_MaxAngularVelocity_RadPerS,
        AngularVelocity_RadPerS + AngularAccel_RadPerS2 * CycleTime_S, CST_MaxAngularVelocity_RadPerS);
    Angle_Rad := LIMIT(-CST_MaxAngle_Rad, Angle_Rad + AngularVelocity_RadPerS * CycleTime_S,
        CST_MaxAngle_Rad);
    IF BrakeMechanicallyOpen THEN
        VelocityReaction_Mps := ReactionGain_Mps2 * Angle_Rad * CycleTime_S;
    END_IF;
END_IF;
Ready := TRUE;

          
END_FUNCTION_BLOCK

(* DOC: DOC/AF/AF_Partie-13_Fonction_Simulation_v2.5.md Chaine bobine, effet mecanique et contact frein M3. *)
FUNCTION_BLOCK FB_Sim_TranslationBrake
  VAR_INPUT
    Enable : BOOL;
    ReleaseCmd : BOOL;
    ActualFrequency_Hz : REAL;
    OpenDelay_S : REAL := 0.1;
    CloseDelay_S : REAL := 0.09;
    ContactDelay_S : REAL := 0.01;
    CycleTime_S : REAL := 0.01;
    FaultCloseWhileRunning : BOOL := FALSE;  (* Branche de FAUTE EXPLICITE — defaut FALSE : chemin nominal strictement inchange. Rejoue le defaut terrain « cause 6 instantanee » : contact frein ferme alors que le variateur retourne encore de la vitesse (trace 2026-09-04, 26,437 s, 10,00 Hz, State.ErrorId=64). La garde nominale CST_StopFrequency_Hz est CONSERVEE telle quelle : elle est validee par la meme trace (frein ouvert a 0,60 Hz, ferme a 0,00 Hz). *)
    FaultCloseDelay_S : REAL := 0;
    PhysicalBrakeActive : BOOL := FALSE;  (* L3 — FREIN PHYSIQUE (2026-10-28). FALSE = historique : la retombee mecanique attend f <= 0,5 Hz (garde qui recopiait la logique PLC dans l'usine simulee). TRUE = frein a manque de courant reel : retombe CloseDelay_S apres la coupure bobine, QUELLE QUE SOIT la vitesse. defaut FB = historique ; la simulation M3 passe TRUE via GVL_Simulation (source unique) *)
  END_VAR
  VAR_OUTPUT
    Ready : BOOL;
    CoilEnergized : BOOL;
    MechanicallyOpen : BOOL;
    ContactOpen : BOOL;
    FaultCloseActive : BOOL;  (* <-- [DIAG] Branche de faute effectivement appliquee ce scan *)
  END_VAR
  VAR
    MechanicalTimer_S : REAL;
    ContactTimer_S : REAL;
    FaultTimer_S : REAL;
    CST_StopFrequency_Hz : REAL := 0.5;
  END_VAR

            

IF NOT Enable THEN
    Ready := FALSE;
    CoilEnergized := FALSE;
    MechanicallyOpen := FALSE;
    ContactOpen := FALSE;
    FaultCloseActive := FALSE;
    MechanicalTimer_S := 0.0;
    ContactTimer_S := 0.0;
    FaultTimer_S := 0.0;
    RETURN;
END_IF;

(* Faute explicite : chronometre propre, remis a zero des que le stimulus retombe. *)
IF FaultCloseWhileRunning THEN
    FaultTimer_S := FaultTimer_S + CycleTime_S;
ELSE
    FaultTimer_S := 0.0;
END_IF;
FaultCloseActive := FaultCloseWhileRunning AND (FaultTimer_S >= MAX(0.0, FaultCloseDelay_S));

(* La faute fait retomber la bobine : l'etat electrique publie reste coherent avec la
   fermeture mecanique observee (jamais « bobine energisee ET frein serre »). *)
CoilEnergized := ReleaseCmd AND NOT FaultCloseActive;
IF CoilEnergized THEN
    IF NOT MechanicallyOpen THEN
        MechanicalTimer_S := MechanicalTimer_S + CycleTime_S;
        IF MechanicalTimer_S >= MAX(0.0, OpenDelay_S) THEN
            MechanicallyOpen := TRUE;
            MechanicalTimer_S := 0.0;
        END_IF;
    ELSE
        MechanicalTimer_S := 0.0;
    END_IF;
ELSIF FaultCloseActive OR PhysicalBrakeActive OR (ActualFrequency_Hz <= CST_StopFrequency_Hz) THEN
    IF MechanicallyOpen THEN
        MechanicalTimer_S := MechanicalTimer_S + CycleTime_S;
        IF MechanicalTimer_S >= MAX(0.0, CloseDelay_S) THEN
            MechanicallyOpen := FALSE;
            MechanicalTimer_S := 0.0;
        END_IF;
    ELSE
        MechanicalTimer_S := 0.0;
    END_IF;
ELSE
    MechanicalTimer_S := 0.0;
END_IF;
IF MechanicallyOpen <> ContactOpen THEN
    ContactTimer_S := ContactTimer_S + CycleTime_S;
    IF ContactTimer_S >= MAX(0.0, ContactDelay_S) THEN
        ContactOpen := MechanicallyOpen;
        ContactTimer_S := 0.0;
    END_IF;
ELSE
    ContactTimer_S := 0.0;
END_IF;
Ready := TRUE;

          
END_FUNCTION_BLOCK

(* DOC: DOC/AF/AF_Partie-13_Fonction_Simulation_v2.5.md Dynamique reduite du variateur M3, sans commande metier. *)
FUNCTION_BLOCK FB_Sim_TranslationDrive
  VAR_INPUT
    Enable : BOOL;
    FrequencyTgt_Hz : REAL;
    AccelRate_HzPerS : REAL := 20;
    DecelRate_HzPerS : REAL := 20;  (* Pente d'arret relevee sur trace reelle MES (-20.0 Hz/s) *)
    TimeConstant_S : REAL := 0.03;  (* Reponse dynamique AC600 en boucle fermee (30 ms) *)
    LoadAngularVelocity_RadPerS : REAL;
    LoadFrequencyDroopGain_Hz : REAL := 0.5;
    CycleTime_S : REAL := 0.01;
  END_VAR
  VAR_OUTPUT
    Ready : BOOL;
    FrequencyCmd_Hz : REAL;
    ElectricalFrequency_Hz : REAL;
    ActualFrequency_Hz : REAL;
    ResponseAlpha : REAL;
  END_VAR
  VAR
    FrequencyDelta_Hz : REAL;
    FrequencyStep_Hz : REAL;
    CST_MinTime_S : REAL := 0.001;
    CST_StopFrequency_Hz : REAL := 0.5;  (* seuil nominal de fin de rampe variateur *)
    CST_MaxFrequency_Hz : REAL := 50;  (* plafond variateur reel (GVL_PERSISTENT._TranslationMaxFreq_Hz) *)
  END_VAR

            

IF NOT Enable THEN
    Ready := FALSE;
    FrequencyCmd_Hz := 0.0;
    ElectricalFrequency_Hz := 0.0;
    ActualFrequency_Hz := 0.0;
    ResponseAlpha := 0.0;
    RETURN;
END_IF;

FrequencyDelta_Hz := LIMIT(0.0, FrequencyTgt_Hz, CST_MaxFrequency_Hz) - FrequencyCmd_Hz;
IF FrequencyDelta_Hz >= 0.0 THEN
    FrequencyStep_Hz := MAX(0.0, AccelRate_HzPerS) * CycleTime_S;
ELSE
    FrequencyStep_Hz := MAX(0.0, DecelRate_HzPerS) * CycleTime_S;
END_IF;
FrequencyCmd_Hz := FrequencyCmd_Hz + LIMIT(-FrequencyStep_Hz, FrequencyDelta_Hz, FrequencyStep_Hz);
IF TimeConstant_S > CST_MinTime_S THEN
    ResponseAlpha := CycleTime_S / (TimeConstant_S + CycleTime_S);
ELSE
    ResponseAlpha := 1.0;
END_IF;
ElectricalFrequency_Hz := ElectricalFrequency_Hz
    + ResponseAlpha * (FrequencyCmd_Hz - ElectricalFrequency_Hz);
(* Retour AC600 : frequence electrique de sortie. La charge est appliquee par le
   modele mecanique ; elle ne doit pas biaiser le retour publie au PLC. *)
ActualFrequency_Hz := MAX(0.0, ElectricalFrequency_Hz);
IF (FrequencyTgt_Hz <= 0.0) AND (FrequencyCmd_Hz <= 0.0)
    AND (ActualFrequency_Hz <= CST_StopFrequency_Hz) THEN
    ElectricalFrequency_Hz := 0.0;
    ActualFrequency_Hz := 0.0;
END_IF;
Ready := TRUE;

          
END_FUNCTION_BLOCK
